FUNCTION_BLOCK CIRCLE_SET_CURVE_DATA (* Circular movement secondary data *)
  (* Standard: 61499-2 *)
  (* Version 1.0, 02-05-12, GASR, Universidade do Estado de Santa Catarina *)
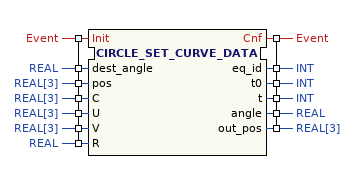
  EVENT_INPUT
    Init WITH dest_angle, pos, C, U, V, R;
  END_EVENT
  EVENT_OUTPUT
    Cnf WITH eq_id, t0, t, angle, out_pos;
  END_EVENT
  VAR_INPUT
    dest_angle : REAL; (* In degrees *)
    pos : ARRAY [0..2] OF REAL;
    C : ARRAY [0..2] OF REAL;
    U : ARRAY [0..2] OF REAL;
    V : ARRAY [0..2] OF REAL;
    R : REAL;
  END_VAR
  VAR_OUTPUT
    eq_id : INT;
    t0 : INT;
    t : INT;
    angle : REAL;
    out_pos : ARRAY [0..2] OF REAL;
  END_VAR
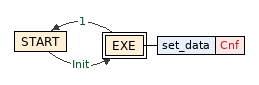
  EC_STATES
    EXE : set_data -> Cnf;
    START;
  END_STATES
  EC_TRANSITIONS
    START TO EXE := Init;
    EXE TO START := 1;
  END_TRANSITIONS
  ALGORITHM set_data IN Lua:
 eq_id = 2 t0 = 0 t = 1 angle = (dest_angle*2*math.pi)/360 out_pos[1] = ( C[1] + U[1]*R*math.cos( angle ) + V[1]*R*math.sin( angle ) ) out_pos[2] = ( C[2] + U[2]*R*math.cos( angle ) + V[2]*R*math.sin( angle ) ) out_pos[3] = ( C[3] + U[3]*R*math.cos( angle ) + V[3]*R*math.sin( angle ) ) print( 'circular_pos', pos[1], pos[2], pos[3], 'circle_destination', out_pos[1], out_pos[2], out_pos[3], 'center'..C[1]..','..C[2]..','..C[3], 'angle', angle ) print( 'circle U',U[1], U[2],U[3], 'circle V', V[1], V[2], V[3], 'radius', R ) print( '\n\n' )
  END_ALGORITHM
END_FUNCTION_BLOCK
